SUBAPPLICATION Uebung_070b (* WBSD auf UT ausgeben, mit QI *)
  (* Standard: 61499-2; Description: Copyright (c) 2023 Meisterschulen am Ostbahnhof This program and the accompanying materials are made available under the terms of the Eclipse Public License 2.0 which is available at https://www.eclipse.org/legal/epl-2.0/ SPDX-License-Identifier: EPL-2.0 *)
  (* Version 1.0, 2023-10-23, Franz Höpfinger, Meisterschulen am Ostbahnhof, initial API and implementation and/or initial documentation *)
  PACKAGE Uebungen;
  IMPORT Uebungen::const::UT::TECU::DefaultPool_TECU::NumberVariable_Wheel_based_machine_speed;
  IMPORT logiBUS::io::DI::logiBUS_DI::Input_I2;
  IMPORT logiBUS::io::DI::logiBUS_DI_Events::BUTTON_SINGLE_CLICK;
  IMPORT logiBUS::io::DQ::logiBUS_DO::Output_Q2;
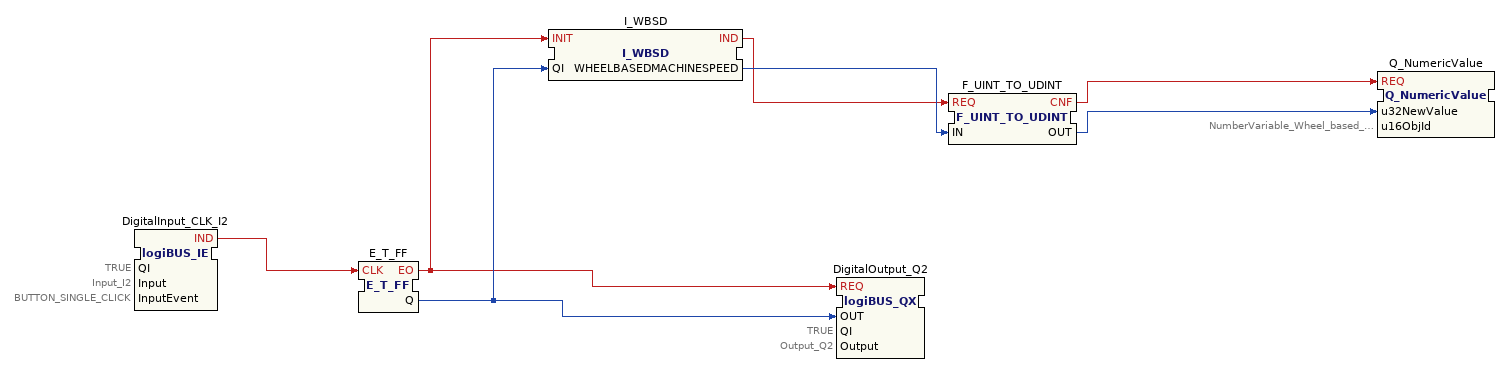
  (* Uebung_094a nutzt dasselbe Prinzip *)
  FBS
    I_WBSD : isobus::tecu::I_WBSD;
    Q_NumericValue : isobus::UT::Q::Q_NumericValue(u16ObjId := NumberVariable_Wheel_based_machine_speed);
    F_UINT_TO_UDINT : iec61131::conversion::F_UINT_TO_UDINT;
    E_T_FF : iec61499::events::E_T_FF;
    DigitalInput_CLK_I2 : logiBUS::io::DI::logiBUS_IE(QI := TRUE, Input := Input_I2, InputEvent := BUTTON_SINGLE_CLICK);
    DigitalOutput_Q2 : logiBUS::io::DQ::logiBUS_QX(QI := TRUE, Output := Output_Q2);
  END_FBS
  EVENT_CONNECTIONS
    F_UINT_TO_UDINT.CNF TO Q_NumericValue.REQ;
    I_WBSD.IND TO F_UINT_TO_UDINT.REQ;
    DigitalInput_CLK_I2.IND TO E_T_FF.CLK;
    E_T_FF.EO TO I_WBSD.INIT;
    E_T_FF.EO TO DigitalOutput_Q2.REQ;
  END_CONNECTIONS
  DATA_CONNECTIONS
    F_UINT_TO_UDINT.OUT TO Q_NumericValue.u32NewValue;
    I_WBSD.WHEELBASEDMACHINESPEED TO F_UINT_TO_UDINT.IN;
    E_T_FF.Q TO DigitalOutput_Q2.OUT;
    E_T_FF.Q TO I_WBSD.QI;
  END_CONNECTIONS
END_SUBAPPLICATION
